PROGRAM POU
VAR
END_VAR

END_PROGRAM

(* stored: Version 1.1.0.1, ProductVersion 3.1.4024.12
   POU POU: Id {551b3377-1ec6-454f-804e-673115bac012}, SpecialFunc None *)
